TYPE ST_FSM_Ctrl :
STRUCT
	bEmergency	:	BOOL;		// Emergenza. Deve essere TRUE perchè la macchina possa operare
	bEnable		:	BOOL;		// Abilitazione macchina. Deve essere TRUE perchè la macchina possa operare
END_STRUCT
END_TYPE

(* stored: Version 1.1.0.1
   DUT ST_FSM_Ctrl: Id {3c6a414a-59ce-0db7-244b-ad031b924eff} *)
